(* Schneider Machine Expert - Basic project Y=A'BC'+DE'F, file version 2.9.0.0 *)
(* ProjectInformations: Name=New project *)

HARDWARE
  Cpu 0: TM221CE24R
  EthernetConfiguration: NetworkName=M221, IpAllocationMode=FixedAddress, IpAddress=0.0.0.0, SubnetMask=0.0.0.0
  SerialLineConfiguration: Baud=Baud19200, Parity=ParityEven, DataBits=DataBits8, StopBits=StopBits1, PhysicalMedium=PhysicalMediumRs485, SlaveId=1, Addressing=SlaveAddressing
  MastTask: UsePeriodScanMode=false, PeriodScan=100
  FastTask: Period=255
  CpuBehavior: StartingMode=StartAsPreviousState, AutoSaveRamOnEeprom=true, WatchdogPeriod=250

SYMBOLS  (address, symbol, comment, settings)
  %I0.0     A
  %I0.1     B
  %I0.2     C
  %I0.3     DS
  %I0.4     ES
  %I0.5     FS
  %Q0.0     Y

POU New POU
  (* SectionNumber=1 *)

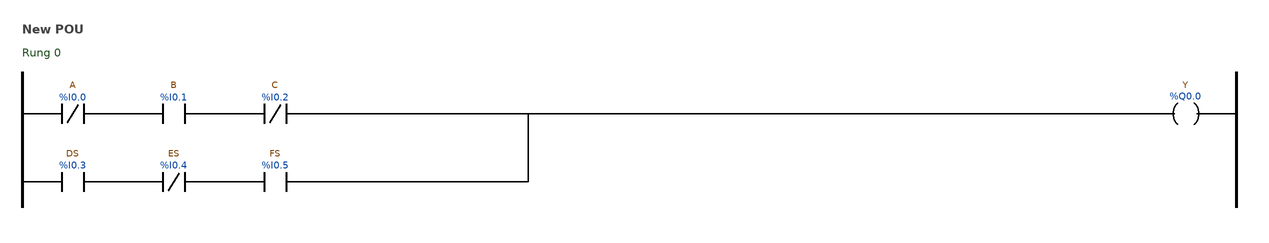

// Rung 0
  LDN %I0.0               (* A *)
  AND %I0.1               (* B *)
  ANDN %I0.2              (* C *)
  OR( %I0.3               (* DS *)
  ANDN %I0.4              (* ES *)
  AND %I0.5               (* FS *)
  )
  ST %Q0.0                (* Y *)
  // as ST:
  //   Y := NOT A AND B AND NOT C OR DS AND NOT ES AND FS;
